Universal Robots PolyScope program: aqw.urp

Program aqw (installation=default directory=/programs createdIn=5.9.1.1031110 lastSavedIn=5.9.1.1031110 robotSerialNumber=20195501059)
Calibrated DH parameters: a=[0.000146, -0.418764, -0.053981, 0.000058, -0.000023, 0]; d=[0.162545, 37.319448, -206.067439, 168.881546, 0.09955, 0.099464]; alpha=[1.57004, -0.001979, 0.002304, 1.570607, -1.57066, 0]; deltaTheta=[0, -0.174616, -1.258233, 1.432844, -0.000001, 0]
BeforeStart
  URCap Gripper Activate (Robotiq_Grippers, Robotiq Inc.) dataModel(ResetAndActivateKey=false)
Robot Program (runOnlyOnce=true)
  URCap Grip Check (Robotiq_Grippers, Robotiq Inc.) dataModel(ObjectDetectedKey=true, DimensionValidationKey=false, DimensionKey=100.0, DimensionDimensionPositiveGapKey=5.0, DimensionNegativeGapKey=5.0, GripperIdKey=1, ModelDefinedKey=true); state(isChildrenLocked=true)
    URCap If (Robotiq_Grippers, Robotiq Inc.)
      Popup Error (haltProgram=false message=Already holding something! inputType=Text)
      Halt
  MoveJ speed 60 deg/s, acceleration 80 deg/s^2 (useActiveTCP=true) feature=Base
    Waypoint Waypoint_1: TCP in base x=234.667 y=-406.867 z=73.131 mm, rx=0.1647 ry=3.1372 rz=-0.0001 rad; joints [103.437, -84.659, 122.188, -127.524, 270.061, 19.478] deg; TCP offset x=0 y=0 z=174 mm, rx=0 ry=0 rz=0 rad
    URCap Gripper (Robotiq_Grippers, Robotiq Inc.) dataModel(position=90.58823529411765, force=100.0, speed=100.0, positionInDouble=90.58823529411765, forceInDouble=100.0, speedInDouble=100.0, slaveIds=[9], blocking=false)
    MoveL speed 250 mm/s, acceleration 1200 mm/s^2 (useActiveTCP=true) feature=Base
      Waypoint nut_pickup: TCP in base x=325.525 y=-452.804 z=18.546 mm, rx=-0.1646 ry=-3.1372 rz=0 rad; joints [111.827, -68.763, 111.567, -132.796, 270.037, 27.874] deg
      MoveDirectionNode (selectedDirection=ZPlus toolParams=0.02, 0.5) feature=Joint_6_name
        Until DISTANCE (allowActions=true deceleration=3 distanceNodeType=STOP) Distance=0.01; motionParameters(blendRadius=0)
          Popup Message (haltProgram=false inputType=Text)
        Until TOOL_CONTACT_DETECTION (allowActions=false retraction=0.001 decelerationAcceleration=3 decelerationAngularAcceleration=34.906585)
      URCap Gripper (Robotiq_Grippers, Robotiq Inc.) dataModel(position=64.31828545371636, force=100.0, speed=100.0, positionInDouble=64.31828545371636, forceInDouble=100.0, speedInDouble=100.0, slaveIds=[9], blocking=true)
      MoveDirectionNode (selectedDirection=ZPlus toolParams=0.02, 0.8) feature=Joint_6_name
        Until TOOL_CONTACT_DETECTION (allowActions=false retraction=0 decelerationAcceleration=3 decelerationAngularAcceleration=34.906585)
      URCap Gripper (Robotiq_Grippers, Robotiq Inc.) dataModel(position=100.0, force=100.0, speed=100.0, positionInDouble=100.0, forceInDouble=100.0, speedInDouble=100.0, slaveIds=[9], blocking=true)
      MoveDirectionNode (selectedDirection=ZPlus) feature=Base
        Until DISTANCE (allowActions=false deceleration=3 distanceNodeType=STOP) Distance=0.01; motionParameters(blendRadius=0)
    MoveL speed 250 mm/s, acceleration 1200 mm/s^2 (useActiveTCP=true) feature=Base
      Waypoint Waypoint_1: TCP in base x=234.667 y=-406.867 z=73.131 mm, rx=0.1647 ry=3.1372 rz=-0.0001 rad; joints [103.437, -84.659, 122.188, -127.524, 270.061, 19.478] deg
